// SIMATIC STEP 7 (V5.x) project MeM840D
// CPU: CPU 314
// station: P_ADR_BUS
// station: Hardware
// station: SIMATIC 300(1)
// program: Programma S7(1)

SYMBOL_TABLE
"POR_SX"	I 34.0	BOOL	// PORTA SX
"POR_DX"	I 34.1	BOOL	// PORTA DX
"CON_AVA"	I 40.4	BOOL	// CONTROPUNTA AVANTI
"CON_IND"	I 40.5	BOOL	// CONTROPUNTA INDIETRO
"BLKMOV"	SFC 20	SFC 20	// Copy Variables
"FILL"	SFC 21	SFC 21	// Initialize a Memory Area
"CREAT_DB"	SFC 22	SFC 22	// Create Data Block
"DIS_AIRT"	SFC 41	SFC 41	// Delay the Higher Priority Interrupts and Asynchronous Errors
"EN_AIRT"	SFC 42	SFC 42	// Enable Higher Priority Interrupts and Asynchronous Errors
"STP"	SFC 46	SFC 46	// Change the CPU to STOP
"WAIT"	SFC 47	SFC 47	// Delay Execution of the User Program
"RDSYSST"	SFC 51	SFC 51	// Read a System Status List or Partial List
"WR_USMSG"	SFC 52	SFC 52	// Write a User-Defined Diagnostic Event to the Diagnostic Buffer
"TIME_TCK"	SFC 64	SFC 64	// Read the System Time
END_SYMBOL_TABLE

// FB 1: know-how protected block, not included

// FB 2: know-how protected block, not included

// FB 3: know-how protected block, not included

// FB 4: know-how protected block, not included

// FB 5: know-how protected block, not included

// FB 6: know-how protected block, not included

// FB 7: know-how protected block, not included

FUNCTION_BLOCK FB 15
VERSION : 0.0
BEGIN
// body was compiled from another editor; compiled code not shown
END_FUNCTION_BLOCK

// FB 16: know-how protected block, not included

// FB 17: know-how protected block, not included

// FB 18: know-how protected block, not included

// FB 19: know-how protected block, not included

FUNCTION_BLOCK FB 20
VERSION : 2.2
BEGIN
// (block stored without names or comments; labels and parameter names are numbered)
NETWORK
TITLE =
      L     DW#16#87000000;
      LAR1;
      L     80;
      L     W#16#A000;
      +I;
      T     LW 0;
      A      [AR1,P#8.0];
      =     L 0.0;
      L     W [AR1,P#0.0];
      T     LW 2;
      L     W [AR1,P#6.0];
      SLD   16;
      L     B [AR1,P#4.0];
      OD;
      T     LD 4;
      CALL  "WR_USMSG" (
           SEND                     := FALSE,
           EVENTN                   := LW 0,
           INFO1                    := P#L 2.0 INT 1,
           INFO2                    := P#L 4.0 DINT 1,
           RET_VAL                  := LW 8);
END_FUNCTION_BLOCK

// FB 28: know-how protected block, not included

FUNCTION_BLOCK FB 120
AUTHOR : USER
VERSION : 0.2
BEGIN
// (block stored without names or comments; labels and parameter names are numbered)
NETWORK
TITLE =
      A     DIX [AR2,P#0.0];
      S     DIX [AR2,P#8.0];
      S     DIX [AR2,P#12.0];
NETWORK
TITLE =
      CALL  FB 3 , DB 91 (
           DIX 0.0                  := DBX [AR2,P#8.0],
           DIW 2                    := 1,
           DIW 4                    := W#16#1002,
           DIW 6                    := 10,
           DIW 8                    := 70,
           DID 10                   := P#DBX 0.0,
           DIX 132.0                := DBX [AR2,P#8.1],
           DIX 132.1                := DBX [AR2,P#8.2],
           DIX 134.0                := DBW [AR2,P#10.0],
           DIW 136                  := W#16#1001,
           DIW 138                  := 1,
           DIW 140                  := DBNO,
           DID 142                  := DBNO);
      A     DIX [AR2,P#8.1];
      =     DIX [AR2,P#2.0];
      R     DIX [AR2,P#8.0];
      A     DIX [AR2,P#8.2];
      =     DIX [AR2,P#2.1];
      R     DIX [AR2,P#8.0];
      L     DIW [AR2,P#10.0];
      T     DIW [AR2,P#4.0];
      A     DIX [AR2,P#8.2];
      AN    DB10.DBX 106.1;
      O     M 110.3;
      L     S5T#500MS;
      SP    T 121;
      A     T 121;
      =     M 110.3;
      A     M 110.3;
      FN    M 110.4;
      S     DIX [AR2,P#6.0];
      A     DB21.DBX 35.7;
      FP    M 110.6;
      A     M 110.6;
      R     DIX [AR2,P#6.0];
NETWORK
TITLE =
      AN    DIX [AR2,P#12.0];
      JC    M002;
      L     W#16#4C;
      +     1;
      T     DIW [AR2,P#14.0];
      OPN   DB 82;
      L     W#16#0;
      SLD   3;
      LAR1;
M001: L     W#16#0;
      T     DBB [AR1,P#0.0];
      +AR1  P#1.0;
      L     DIW [AR2,P#14.0];
      +     -1;
      T     DIW [AR2,P#14.0];
      LOOP  M001;
      SET;
      S     DB82.DBX 4.0;
      S     DB82.DBX 6.0;
      S     DB82.DBX 8.0;
      S     DB82.DBX 10.0;
      R     DIX [AR2,P#12.0];
M002: BE;
END_FUNCTION_BLOCK

// FC 1: know-how protected block, not included

// FC 2: know-how protected block, not included

// FC 3: know-how protected block, not included

// FC 4: know-how protected block, not included

// FC 6: know-how protected block, not included

// FC 7: know-how protected block, not included

// FC 8: know-how protected block, not included

// FC 9: know-how protected block, not included

// FC 10: know-how protected block, not included

// FC 11: know-how protected block, not included

FUNCTION FC 12 : VOID
AUTHOR : NUMERIK
FAMILY : _800D
NAME : Basics
VERSION : 4.0
BEGIN
// (block stored without names or comments; labels and parameter names are numbered)
END_FUNCTION

// FC 13: know-how protected block, not included

// FC 14: know-how protected block, not included

// FC 15: know-how protected block, not included

// FC 16: know-how protected block, not included

// FC 17: know-how protected block, not included

// FC 18: know-how protected block, not included

FUNCTION FC 19 : VOID
AUTHOR : NUMERIK
FAMILY : _800D
NAME : MCP_IFM
VERSION : 5.1
BEGIN
// (block stored without names or comments; labels and parameter names are numbered)
NETWORK
TITLE =
// (network holds code this reader does not know; not shown)
END_FUNCTION

// FC 20: know-how protected block, not included

// FC 21: know-how protected block, not included

// FC 22: know-how protected block, not included

FUNCTION FC 24 : VOID
AUTHOR : NUMERIK
FAMILY : _800D
NAME : MCP_IFM2
VERSION : 5.1
BEGIN
// (block stored without names or comments; labels and parameter names are numbered)
NETWORK
TITLE =
// (network holds code this reader does not know; not shown)
END_FUNCTION

FUNCTION FC 25 : VOID
AUTHOR : NUMERIK
FAMILY : _800D
NAME : MCP_IFT
VERSION : 5.1
BEGIN
// (block stored without names or comments; labels and parameter names are numbered)
NETWORK
TITLE =
// (network holds code this reader does not know; not shown)
END_FUNCTION

FUNCTION FC 26 : VOID
AUTHOR : NUMERIK
FAMILY : _800D
NAME : HPU_MCP
VERSION : 6.1
BEGIN
// (block stored without names or comments; labels and parameter names are numbered)
NETWORK
TITLE =
// (network holds code this reader does not know; not shown)
END_FUNCTION

FUNCTION FC 30 : VOID
VERSION : 0.0
BEGIN
// body was compiled from another editor; compiled code not shown
END_FUNCTION

FUNCTION FC 31 : VOID
VERSION : 0.0
BEGIN
// body was compiled from another editor; compiled code not shown
END_FUNCTION

FUNCTION FC 32 : VOID
VERSION : 0.0
BEGIN
// body was compiled from another editor; compiled code not shown
END_FUNCTION

FUNCTION FC 33 : VOID
VERSION : 0.0
BEGIN
// body was compiled from another editor; compiled code not shown
END_FUNCTION

// FC 34: know-how protected block, not included

// FC 35: know-how protected block, not included

FUNCTION FC 52 : VOID
AUTHOR : Zagorski
NAME : GENFUNK
VERSION : 0.15
BEGIN
// (block stored without names or comments; labels and parameter names are numbered)
NETWORK
TITLE =
      A     I 33.0;
      =     DB31.DBX 12.7;
      A     M 129.1;
      JC    M001;
      A     I 33.1;
      A     DB32.DBX 64.7;
      FN    M 15.0;
      =     M 15.1;
      A     I 33.1;
      S     M 15.2;
      A     M 15.1;
      R     M 15.2;
      A     M 15.2;
      =     DB32.DBX 12.7;
      JU    M002;
M001: A     I 6.7;
      A     I 2.7;
      AN    M 16.4;
      =     M 16.5;
      A     I 6.7;
      A     I 2.7;
      =     M 16.4;
      A     M 16.5;
      A     Q 4.7;
      R     M 16.6;
      A     M 16.5;
      AN    Q 4.7;
      S     M 16.6;
      A     M 16.6;
      =     Q 4.7;
      A     M 16.6;
      =     DB32.DBX 2.5;
      A     M 16.6;
      S     M 16.7;
      A     DB32.DBX 60.4;
      ON    M 16.6;
      R     M 16.7;
      L     PIW 32;
      T     MW 17;
      L     PIB 34;
      T     MB 19;
      A     M 18.1;
      A     DB32.DBX 64.7;
      FN    M 15.0;
      =     M 15.1;
      A     M 18.1;
      S     M 15.2;
      A     M 15.1;
      R     M 15.2;
      A     M 19.5;
      A     DB32.DBX 64.7;
      FN    M 15.4;
      =     M 15.5;
      A     M 19.5;
      S     M 15.6;
      A     M 15.5;
      R     M 15.6;
      A     M 16.6;
      A     M 15.6;
      O;
      AN    M 16.6;
      A     M 15.2;
      =     DB32.DBX 12.7;
M002: O     I 3.7;
      ON    I 32.0;
      =     M 75.1;
      O     I 3.7;
      ON    I 32.0;
      =     M 75.1;
      A     DB10.DBX 108.7;
      A(;
      O     I 32.0;
      O;
      A     I 3.7;
      A     I 4.4;
      A     Q 4.3;
      A     Q 0.4;
      );
      =     Q 36.4;
      A     DB10.DBX 108.7;
      =     Q 36.0;
      AN    I 32.0;
      A(;
      ON    I 3.7;
      ON    I 4.4;
      ON    Q 4.3;
      ON    Q 0.4;
      );
      =     DB10.DBX 56.1;
      A     I 32.0;
      O(;
      A     I 3.7;
      A     I 4.4;
      A     Q 4.3;
      A     Q 0.4;
      );
      AN    DB10.DBX 56.1;
      =     DB10.DBX 56.2;
NETWORK
TITLE =
      A     I 32.0;
      A     M 39.0;
      O;
      AN    DB33.DBX 61.4;
      A(;
      ON    M 39.0;
      ON    I 32.0;
      );
      O;
      A     I 3.7;
      A     I 4.4;
      A     Q 4.3;
      A     Q 0.4;
      =     DB31.DBX 2.1;
      =     DB31.DBX 21.7;
      =     DB32.DBX 2.1;
      =     DB32.DBX 21.7;
      =     DB33.DBX 2.1;
      =     DB33.DBX 21.7;
      A     M 51.0;
      =     DB21.DBX 25.3;
      =     DB31.DBX 1.5;
      =     DB32.DBX 1.5;
      =     DB33.DBX 1.6;
NETWORK
TITLE =
      A     I 5.5;
      A(;
      O     I 3.6;
      O     I 4.4;
      );
      =     M 40.4;
NETWORK
TITLE =
      A     M 40.4;
      A(;
      O     I 32.0;
      O;
      A     I 3.7;
      A     I 4.4;
      A     Q 4.3;
      A     Q 0.4;
      );
      S     M 39.0;
NETWORK
TITLE =
      O;
      A     I 4.2;
      A     DB33.DBX 61.4;
      AN    DB21.DBX 35.5;
      AN    DB21.DBX 35.0;
      O;
      AN    I 32.0;
      A(;
      ON    I 3.7;
      ON    I 4.4;
      ON    Q 4.3;
      ON    Q 0.4;
      );
      O     M 75.2;
      R     M 39.0;
NETWORK
TITLE =
      A     M 39.0;
      =     Q 3.6;
      AN    M 39.0;
      =     Q 2.5;
NETWORK
TITLE =
      A     M 39.0;
      A     I 32.0;
      O;
      A     I 3.7;
      A     I 4.4;
      A     Q 4.3;
      A     Q 0.4;
      S     Q 37.7;
      A     DB33.DBX 61.4;
      A(;
      ON    M 39.0;
      ON    I 32.0;
      );
      A(;
      ON    I 3.7;
      ON    I 4.4;
      ON    Q 4.3;
      ON    Q 0.4;
      );
      R     Q 37.7;
NETWORK
TITLE =
      A     I 32.0;
      FN    M 3.1;
      =     M 3.2;
      A     M 3.2;
      S     M 3.0;
      A     I 3.7;
      R     M 3.0;
NETWORK
TITLE =
      L     DB82.DBB 45;
      L     0;
      ==I;
      =     M 38.0;
NETWORK
TITLE =
      L     DB82.DBB 45;
      L     3;
      <=I;
      =     M 38.6;
NETWORK
TITLE =
      A     DB33.DBX 82.3;
      =     DB82.DBX 16.6;
      A     DB33.DBX 82.3;
      A     DB33.DBX 61.4;
      S     M 40.0;
      A     DB33.DBX 16.3;
      R     M 40.0;
      A     M 40.0;
      =     DB33.DBX 18.5;
      AN    M 40.0;
      JC    M003;
      A     DB33.DBX 82.0;
      AN    DB33.DBX 82.1;
      AN    DB33.DBX 82.2;
      S     Q 36.1;
      R     Q 36.2;
      AN    DB33.DBX 82.0;
      A     DB33.DBX 82.1;
      AN    DB33.DBX 82.2;
      S     Q 36.2;
      R     Q 36.1;
M003: A     I 33.6;
      AN    I 33.7;
      S     DB33.DBX 16.0;
      R     DB33.DBX 16.1;
      R     DB33.DBX 16.2;
      AN    I 33.6;
      A     I 33.7;
      R     DB33.DBX 16.0;
      S     DB33.DBX 16.1;
      R     DB33.DBX 16.2;
      A     DB33.DBX 16.0;
      =     M 41.0;
      A     DB33.DBX 16.1;
      =     M 41.1;
      A     DB33.DBX 16.2;
      =     M 41.2;
      A     DB33.DBX 82.0;
      =     M 42.0;
      A     DB33.DBX 82.1;
      =     M 42.1;
      A     DB33.DBX 82.2;
      =     M 42.2;
      L     MB 41;
      L     MB 42;
      ==I;
      =     M 40.1;
      A     M 40.1;
      L     S5T#2S;
      SD    T 70;
      A     T 70;
      =     M 40.2;
      A     M 40.2;
      A     M 40.0;
      S     M 40.3;
      AN    M 40.0;
      R     M 40.3;
      A     M 40.3;
      =     DB33.DBX 16.3;
      AN    M 40.0;
      L     S5T#4S;
      SP    T 69;
NETWORK
TITLE =
      O     I 7.1;
      AN    DB21.DBX 35.0;
      AN    DB21.DBX 35.1;
      =     DB33.DBX 4.7;
      =     Q 5.1;
      AN    I 7.1;
      L     S5T#4S;
      SP    T 68;
NETWORK
TITLE =
      A     I 3.7;
      A     I 4.4;
      A     Q 4.3;
      A     Q 0.4;
      A(;
      A     DB82.DBX 40.0;
      A     M 38.0;
      O;
      AN    DB82.DBX 40.0;
      A     DB11.DBX 6.2;
      );
      =     Q 37.3;
NETWORK
TITLE =
      A     DB33.DBX 61.4;
      L     S5T#4S;
      SF    T 55;
      NOP   0;
      NOP   0;
      NOP   0;
      NOP   0;
NETWORK
TITLE =
      A(;
      O     Q 5.1;
      O     T 68;
      O     M 40.0;
      O     T 69;
      );
      A(;
      A     DB82.DBX 40.0;
      AN    DB82.DBX 41.5;
      O;
      AN    DB82.DBX 40.0;
      AN    DB21.DBX 35.0;
      );
      O;
      A(;
      A(;
      A     DB82.DBX 40.0;
      A     M 38.0;
      O;
      AN    DB82.DBX 40.0;
      A(;
      O     DB11.DBX 6.2;
      O     DB11.DBX 7.2;
      O     DB11.DBX 6.1;
      );
      O;
      A     T 55;
      A(;
      A     DB82.DBX 40.0;
      AN    DB82.DBX 41.5;
      O;
      AN    DB82.DBX 40.0;
      AN    DB21.DBX 35.0;
      O     DB21.DBX 33.7;
      O     DB21.DBX 33.4;
      O;
      A     DB82.DBX 40.0;
      A     DB82.DBX 41.6;
      A     Q 1.4;
      A     Q 1.6;
      A(;
      O     Q 2.0;
      O     Q 3.4;
      );
      O;
      A     DB82.DBX 40.0;
      A     DB82.DBX 41.6;
      A     DB21.DBX 32.5;
      A     Q 1.4;
      O;
      AN    DB82.DBX 40.0;
      A     DB21.DBX 35.2;
      A     Q 1.4;
      A     Q 1.6;
      A     Q 2.0;
      );
      );
      AN    M 3.0;
      O;
      A     I 3.7;
      A     M 3.0;
      );
      A(;
      O     Q 2.0;
      O     Q 3.4;
      O;
      A     DB33.DBX 61.4;
      A     DB21.DBX 32.5;
      );
      =     Q 37.4;
NETWORK
TITLE =
NETWORK
TITLE =
      A(;
      A     DB82.DBX 40.0;
      A     M 38.0;
      O;
      AN    DB82.DBX 40.0;
      A     DB11.DBX 6.2;
      );
      A     I 4.4;
      =     M 16.1;
NETWORK
TITLE =
      AN    "POR_SX";
      AN    "POR_DX";
      AN    I 34.2;
      A(;
      AN    M 45.0;
      AN    M 45.1;
      O     M 134.0;
      O     M 134.1;
      );
      JC    M004;
      A     M 51.0;
      AN    Q 5.1;
      AN    M 40.0;
      S     DB33.DBX 4.3;
      S     DB82.DBX 10.1;
      R     DB82.DBX 10.0;
      AN    Q 5.1;
      AN    M 40.0;
      AN    DB21.DBX 32.5;
      R     I 2.4;
      A     DB33.DBX 61.4;
      AN    Q 5.1;
      AN    M 40.0;
      S     M 71.0;
      A     M 71.0;
      AN    Q 5.1;
      AN    T 68;
      AN    M 40.0;
      AN    T 69;
      R     DB33.DBX 21.7;
M004: AN    "POR_SX";
      AN    "POR_DX";
      AN    I 34.2;
      A(;
      AN    M 45.0;
      AN    M 45.1;
      O     M 134.0;
      O     M 134.1;
      );
      R     M 71.0;
NETWORK
TITLE =
      AN    "POR_SX";
      AN    "POR_DX";
      A(;
      ON    DB33.DBX 61.4;
      O;
      A(;
      A     DB82.DBX 40.0;
      AN    M 38.0;
      O;
      AN    DB82.DBX 40.0;
      AN    DB11.DBX 6.2;
      AN    DB11.DBX 7.2;
      AN    DB11.DBX 6.1;
      );
      A(;
      O     DB21.DBX 35.5;
      O     DB21.DBX 35.0;
      );
      O;
      A     DB82.DBX 40.0;
      AN    M 38.0;
      A     DB82.DBX 41.6;
      AN    DB21.DBX 32.5;
      A(;
      ON    Q 1.4;
      ON    Q 1.6;
      O;
      AN    Q 2.0;
      AN    Q 3.4;
      );
      O;
      AN    DB82.DBX 40.0;
      AN    DB11.DBX 6.2;
      AN    DB11.DBX 7.2;
      AN    DB11.DBX 6.1;
      A     DB21.DBX 35.2;
      AN    DB21.DBX 32.5;
      A(;
      ON    Q 1.4;
      ON    Q 1.6;
      ON    Q 2.0;
      );
      );
      =     Q 36.3;
NETWORK
TITLE =
      AN    DB82.DBX 40.0;
      A     I 3.7;
      =     DB33.DBX 2.2;
NETWORK
TITLE =
      O     "POR_SX";
      O     "POR_DX";
      A(;
      A     DB82.DBX 40.0;
      AN    M 38.6;
      O;
      AN    DB82.DBX 40.0;
      AN    DB11.DBX 6.2;
      AN    DB11.DBX 7.2;
      AN    DB11.DBX 6.1;
      );
      O     I 34.2;
      =     M 38.7;
      O     M 38.7;
      O;
      AN    I 41.7;
      AN    M 16.1;
      =     DB21.DBX 7.0;
      S     DB21.DBX 6.1;
      S     DB21.DBX 6.0;
      S     DB21.DBX 7.3;
NETWORK
TITLE =
      A     M 126.0;
      JC    M005;
      A     M 76.2;
      AN    M 75.3;
      A(;
      A     DB82.DBX 40.0;
      AN    M 38.0;
      O;
      AN    DB82.DBX 40.0;
      AN    DB11.DBX 6.2;
      AN    DB11.DBX 7.2;
      );
      S     DB21.DBX 6.1;
M005: NOP   0;
NETWORK
TITLE =
      A     M 126.0;
      JC    M006;
      A     M 51.0;
      A     M 76.2;
      AN    M 75.3;
      A(;
      A     DB82.DBX 40.0;
      AN    M 38.0;
      O;
      AN    DB82.DBX 40.0;
      AN    DB11.DBX 6.2;
      AN    DB11.DBX 7.2;
      );
      S     DB21.DBX 6.0;
M006: NOP   0;
NETWORK
TITLE =
      A     I 34.2;
      =     DB2.DBX 180.0;
      A     I 35.4;
      =     DB2.DBX 180.3;
      A     M 12.7;
      =     DB2.DBX 180.5;
      A     T 66;
      =     DB2.DBX 180.6;
      A(;
      O     M 134.2;
      O     M 134.3;
      O     M 134.4;
      );
      A(;
      O     M 45.0;
      O     M 45.1;
      AN    DB33.DBX 4.7;
      AN    M 40.0;
      AN    I 4.4;
      );
      A(;
      ON    DB33.DBX 61.4;
      O     I 2.5;
      O     I 5.4;
      O     I 4.0;
      O     I 2.1;
      );
      =     DB2.DBX 180.7;
      A     M 134.0;
      AN    I 35.0;
      =     DB2.DBX 181.0;
      AN    I 35.1;
      =     DB2.DBX 181.1;
      AN    I 35.2;
      =     DB2.DBX 181.2;
      AN    M 134.0;
      AN    I 35.0;
      =     DB2.DBX 181.3;
      AN    I 35.6;
      =     DB2.DBX 181.4;
      AN    I 35.7;
      =     DB2.DBX 181.5;
      AN    M 125.0;
      AN    I 35.5;
      =     DB2.DBX 181.6;
      AN    M 39.0;
      =     DB2.DBX 185.0;
      AN    M 40.0;
      A(;
      AN    I 33.6;
      AN    I 33.7;
      O;
      A     I 33.6;
      A     I 33.7;
      );
      =     DB2.DBX 185.2;
      JU    M007;
      A(;
      O     "POR_SX";
      O     "POR_DX";
      );
      A(;
      A     DB82.DBX 40.0;
      AN    M 38.6;
      O;
      AN    DB82.DBX 40.0;
      AN    DB11.DBX 6.2;
      AN    DB11.DBX 7.2;
      AN    DB11.DBX 6.1;
      );
      A(;
      O     I 2.5;
      O     I 5.4;
      O     I 4.0;
      O     I 2.1;
      );
      S     M 15.3;
      A(;
      AN    "POR_SX";
      AN    "POR_DX";
      O;
      A     DB82.DBX 40.0;
      A     M 38.6;
      O;
      AN    DB82.DBX 40.0;
      A(;
      O     DB11.DBX 6.2;
      O     DB11.DBX 7.2;
      O     DB11.DBX 6.1;
      );
      );
      O     M 75.1;
      O     I 2.4;
      O     I 5.3;
      R     M 15.3;
      A     "POR_SX";
      A(;
      O     M 10.3;
      ON    M 38.7;
      );
      A     M 15.3;
      A(;
      A     DB82.DBX 40.0;
      AN    M 38.6;
      O;
      AN    DB82.DBX 40.0;
      AN    DB11.DBX 6.2;
      AN    DB11.DBX 7.2;
      AN    DB11.DBX 6.1;
      );
      =     DB2.DBX 185.3;
      A     "POR_DX";
      A(;
      O     M 10.3;
      ON    M 38.7;
      );
      A     M 15.3;
      A(;
      A     DB82.DBX 40.0;
      AN    M 38.6;
      O;
      AN    DB82.DBX 40.0;
      AN    DB11.DBX 6.2;
      AN    DB11.DBX 7.2;
      AN    DB11.DBX 6.1;
      );
      =     DB2.DBX 185.4;
      A     M 38.7;
      AN    M 10.3;
      A     M 15.3;
      =     DB2.DBX 185.5;
M007: NOP   0;
      A(;
      O     "POR_SX";
      O     "POR_DX";
      );
      A(;
      O     I 2.5;
      O     I 5.4;
      O     I 4.0;
      O     I 2.1;
      );
      S     M 15.3;
      AN    "POR_SX";
      AN    "POR_DX";
      O     M 75.1;
      O     I 2.4;
      O     I 5.3;
      R     M 15.3;
      A     "POR_SX";
      A(;
      O     M 10.3;
      ON    M 38.7;
      );
      A     M 15.3;
      =     DB2.DBX 185.3;
      A     "POR_DX";
      A(;
      O     M 10.3;
      ON    M 38.7;
      );
      A     M 15.3;
      =     DB2.DBX 185.4;
      A     M 38.7;
      AN    M 10.3;
      A     M 15.3;
      =     DB2.DBX 185.5;
      A     M 126.0;
      JC    M008;
      A     M 76.3;
      =     DB2.DBX 180.1;
      A     M 76.7;
      =     DB2.DBX 180.2;
      A(;
      O     Q 37.0;
      O     Q 37.1;
      );
      A     I 33.3;
      L     S5T#80MS;
      SD    T 87;
      NOP   0;
      NOP   0;
      NOP   0;
      NOP   0;
      A     I 32.0;
      A     T 87;
      S     M 76.6;
      A     M 75.1;
      R     M 76.6;
      A     M 76.6;
      =     DB2.DBX 185.7;
      A     M 75.4;
      AN    M 77.4;
      =     DB2.DBX 186.0;
      A     M 77.5;
      =     DB2.DBX 186.1;
      AN    M 88.4;
      AN    M 77.5;
      AN    T 87;
      =     DB2.DBX 186.2;
      AN    M 77.4;
      AN    M 75.4;
      AN    M 77.5;
      AN    T 87;
      =     DB2.DBX 186.3;
M008: NOP   0;
      A     M 129.1;
      A     M 16.7;
      =     DB2.DBX 186.4;
      A(;
      O     M 134.2;
      O     M 134.4;
      );
      A(;
      A     Q 38.6;
      A     M 46.7;
      O;
      A     Q 38.5;
      AN    M 46.7;
      );
      =     DB2.DBX 186.5;
      A(;
      O     M 134.3;
      O     M 134.4;
      );
      A     Q 38.3;
      AN    M 44.0;
      =     DB2.DBX 186.6;
      A(;
      O     M 134.2;
      O     M 134.4;
      );
      AN    M 45.4;
      A(;
      O     I 40.0;
      O     I 40.1;
      );
      O;
      A(;
      O     M 134.3;
      O     M 134.4;
      );
      AN    M 45.5;
      A(;
      O     "CON_AVA";
      O     "CON_IND";
      );
      =     DB2.DBX 186.7;
      A(;
      O     M 134.2;
      O     M 134.4;
      );
      A(;
      A     Q 38.5;
      AN    Q 38.6;
      AN    I 34.6;
      );
      A     Q 36.4;
      =     DB2.DBX 187.0;
      A(;
      O     M 134.3;
      O     M 134.4;
      );
      AN    I 41.0;
      A     Q 38.0;
      A     Q 36.4;
      =     DB2.DBX 187.1;
      A(;
      O     M 134.2;
      O     M 134.4;
      );
      A     M 45.1;
      =     DB2.DBX 187.2;
      JU    M009;
      A     M 72.1;
      A     M 72.0;
      L     S5T#4S;
      SD    T 73;
      A     T 73;
      =     DB2.DBX 187.3;
      AN    M 72.1;
      A     M 72.0;
      L     S5T#4S;
      SD    T 74;
      A     T 74;
      =     DB2.DBX 187.4;
M009: NOP   0;
      AN    I 32.1;
      A     M 39.0;
      =     DB2.DBX 192.0;
      AN    I 41.7;
      =     DB2.DBX 194.0;
      A(;
      ON    M 43.7;
      O     M 43.5;
      ON    DB11.DBX 6.2;
      O     DB21.DBX 35.0;
      O     DB21.DBX 35.1;
      );
      A     I 4.4;
      A     I 6.7;
      =     DB2.DBX 194.4;
NETWORK
TITLE =
      A     M 75.2;
      R     M 10.0;
      R     M 10.2;
      R     M 10.6;
      O(;
      A     DB31.DBX 76.0;
      FN    M 11.0;
      );
      O(;
      A     DB31.DBX 76.0;
      FP    M 11.1;
      );
      =     M 11.2;
      O(;
      A     DB32.DBX 76.0;
      FN    M 10.4;
      );
      O(;
      A     DB32.DBX 76.0;
      FP    M 10.5;
      );
      =     M 10.7;
      AN    M 10.6;
      L     S5T#2S;
      SD    T 64;
      A     T 64;
      =     M 10.6;
      A     M 10.0;
      O     M 11.2;
      O     M 10.7;
      L     C#600;
      S     C 1;
      A     M 10.6;
      A     DB31.DBX 61.4;
      A     DB32.DBX 61.4;
      CD    C 1;
      L     C 1;
      L     0;
      ==I;
      =     M 10.0;
      A     M 10.0;
      O     M 11.2;
      O     M 10.7;
      L     S5T#10S;
      SE    T 61;
      A     T 61;
      =     M 10.1;
      AN    M 10.2;
      L     S5T#4S;
      SE    T 62;
      A     T 62;
      =     M 10.2;
      A     M 10.2;
      L     S5T#2S;
      SE    T 63;
      A     T 63;
      =     M 10.3;
      A     M 10.1;
      A     M 10.6;
      AN    M 14.5;
      S     M 14.2;
      O     M 14.4;
      O     T 59;
      O;
      A     M 12.7;
      A(;
      O     M 75.1;
      O     M 75.2;
      );
      R     M 14.2;
      A     M 14.2;
      A     I 35.3;
      L     S5T#1S;
      SE    T 60;
      A     T 60;
      FN    M 14.3;
      =     M 14.4;
      A     M 14.4;
      S     M 14.5;
      A     T 59;
      R     M 14.5;
      A     M 14.5;
      AN    I 35.3;
      L     S5T#1S;
      SE    T 59;
      A     I 7.7;
      AN    I 35.3;
      S     M 14.0;
      A     M 14.0;
      A     I 7.7;
      A     I 35.3;
      S     M 14.1;
      A     M 14.0;
      A     M 14.1;
      L     S5T#2S;
      SE    T 67;
      O     T 67;
      ON    I 7.7;
      R     M 14.0;
      R     M 14.1;
      A(;
      A     M 14.2;
      A(;
      O     M 10.1;
      ON    M 14.2;
      ON    M 12.7;
      );
      O;
      AN    I 35.3;
      A     I 7.7;
      AN    T 67;
      );
      A     I 32.0;
      =     Q 36.6;
      =     Q 5.7;
      A     M 10.1;
      A     I 35.3;
      FN    M 11.4;
      =     M 11.5;
      A     M 10.1;
      A     I 35.3;
      FP    M 11.6;
      =     M 11.7;
      A     M 10.1;
      A     Q 36.6;
      FN    M 12.0;
      =     M 12.1;
      A     M 10.1;
      A     Q 36.6;
      FP    M 12.2;
      =     M 12.3;
      AN    I 7.7;
      A(;
      O     M 12.1;
      O     M 12.3;
      );
      AN    M 12.4;
      S     M 12.5;
      AN    I 7.7;
      A(;
      O     M 11.5;
      O     M 11.7;
      );
      A     M 12.4;
      S     M 12.6;
      O     M 12.1;
      O     M 12.3;
      S     M 12.4;
      AN    M 10.1;
      AN    Q 36.6;
      R     M 12.4;
      A     M 12.5;
      A     M 12.6;
      AN    M 10.1;
      A     M 10.3;
      O     M 75.1;
      O     M 75.2;
      R     M 12.4;
      R     M 12.5;
      R     M 12.6;
      R     M 12.7;
      A     M 12.5;
      AN    M 12.6;
      AN    M 10.1;
      S     M 12.7;
NETWORK
TITLE =
      A     Q 36.4;
      A     I 35.0;
      L     S5T#5S;
      SD    T 65;
      AN    I 34.3;
      A     T 65;
      L     S5T#5S;
      SD    T 66;
NETWORK
TITLE =
      A     I 7.5;
      AN    M 70.0;
      =     M 70.1;
      A     I 7.5;
      =     M 70.0;
      A     M 70.1;
      O     DB21.DBX 195.1;
      O     DB21.DBX 197.6;
      A     Q 36.5;
      ON    I 32.0;
      R     M 70.2;
      A     M 70.1;
      O     DB21.DBX 194.7;
      A     I 32.0;
      AN    Q 36.5;
      S     M 70.2;
      A     M 70.2;
      A     I 35.1;
      =     Q 36.5;
      =     Q 5.5;
NETWORK
TITLE =
      A     M 125.0;
      JC    M010;
      CALL  FC 70;
M010: NOP   0;
NETWORK
TITLE =
      A     I 5.0;
      AN    M 70.4;
      =     M 70.5;
      A     I 5.0;
      =     M 70.4;
      A     M 70.5;
      A     Q 37.6;
      R     M 70.6;
      A     M 70.5;
      AN    Q 37.6;
      S     M 70.6;
      A     M 70.6;
      =     Q 37.6;
      =     Q 3.1;
NETWORK
TITLE =
      A     DB82.DBX 40.0;
      AN    DB33.DBX 94.6;
      A     DB21.DBX 316.0;
      FN    M 111.0;
      S     DB2.DBX 145.0;
      A     DB33.DBX 83.5;
      R     DB2.DBX 145.0;
      A     DB2.DBX 145.0;
      S     DB21.DBX 6.0;
NETWORK
TITLE =
NETWORK
TITLE =
      AN    DB82.DBX 40.0;
      S     DB10.DBX 57.0;
END_FUNCTION

FUNCTION FC 60 : VOID
AUTHOR : ZAGORSKI
NAME : HYDRCS
VERSION : 0.2
BEGIN
// (block stored without names or comments; labels and parameter names are numbered)
NETWORK
TITLE =
      A     M 134.0;
      JC    M001;
NETWORK
TITLE =
      A     I 34.4;
      A     M 39.0;
      =     M 39.4;
NETWORK
TITLE =
      A     I 5.5;
      A(;
      O     I 3.6;
      O     I 4.4;
      );
      =     M 40.4;
NETWORK
TITLE =
      A     M 40.4;
      A     M 51.0;
      A(;
      O     I 32.0;
      O;
      A     I 3.7;
      A     I 4.4;
      A     Q 4.3;
      A     Q 0.4;
      );
      S     M 39.0;
NETWORK
TITLE =
      AN    M 39.4;
      L     S5T#1S;
      SD    T 35;
      NOP   0;
      NOP   0;
      NOP   0;
      NOP   0;
NETWORK
TITLE =
      A     M 39.0;
      L     S5T#5S;
      SP    T 30;
      NOP   0;
      NOP   0;
      NOP   0;
      NOP   0;
NETWORK
TITLE =
      A(;
      A     I 4.2;
      A     DB33.DBX 61.4;
      AN    DB21.DBX 35.5;
      AN    DB21.DBX 35.0;
      O;
      AN    I 32.0;
      A(;
      ON    I 3.7;
      ON    I 4.4;
      ON    Q 4.3;
      ON    Q 0.4;
      );
      O     M 75.2;
      ON    I 35.0;
      O;
      AN    T 30;
      A     T 35;
      );
      R     M 39.0;
      NOP   0;
      NOP   0;
NETWORK
TITLE =
      A     M 39.0;
      =     Q 36.4;
      =     Q 3.6;
      AN    M 39.0;
      =     Q 2.5;
NETWORK
TITLE =
M001: NOP   0;
NETWORK
TITLE =
      A     DB33.DBX 61.4;
      A(;
      O     DB11.DBX 6.2;
      O;
      AN    DB21.DBX 35.0;
      AN    DB21.DBX 35.5;
      A(;
      O     DB11.DBX 6.1;
      O     DB11.DBX 6.0;
      );
      );
      A     M 39.0;
      L     S5T#2S;
      SD    T 31;
      NOP   0;
      NOP   0;
      NOP   0;
      A     T 31;
      =     M 45.7;
NETWORK
TITLE =
      A     M 45.7;
      AN    I 40.0;
      AN    I 40.1;
      S     M 45.4;
      A(;
      ON    M 45.7;
      );
      R     M 45.4;
      NOP   0;
NETWORK
TITLE =
      A     M 45.7;
      AN    "CON_AVA";
      AN    "CON_IND";
      A(;
      O     "POR_SX";
      O     "POR_DX";
      );
      S     M 45.5;
      A(;
      ON    M 45.7;
      O;
      AN    "POR_SX";
      AN    "POR_DX";
      );
      R     M 45.5;
      NOP   0;
NETWORK
TITLE =
      A     I 6.7;
      AN    M 43.1;
      =     M 43.0;
NETWORK
TITLE =
      A     I 6.7;
      =     M 43.1;
NETWORK
TITLE =
      AN    Q 38.5;
      A     Q 38.6;
      A     I 34.4;
      AN    I 34.6;
      AN    I 40.3;
      A     I 40.2;
      A     M 46.7;
      O;
      A     Q 38.5;
      AN    Q 38.6;
      AN    I 34.4;
      A     I 34.6;
      A     I 40.3;
      AN    I 40.2;
      AN    M 46.7;
      =     M 43.7;
NETWORK
TITLE =
      A     Q 38.5;
      AN    Q 38.6;
      AN    I 34.4;
      A     I 34.6;
      A     I 40.3;
      AN    I 40.2;
      A     M 46.7;
      O;
      AN    Q 38.5;
      A     Q 38.6;
      A     I 34.4;
      AN    I 34.6;
      AN    I 40.3;
      A     I 40.2;
      AN    M 46.7;
      =     M 43.5;
NETWORK
TITLE =
      A     DB11.DBX 6.2;
      AN    DB21.DBX 35.0;
      AN    DB21.DBX 35.1;
      A     I 4.4;
      A     M 43.7;
      AN    M 43.5;
      A     M 43.0;
      A     M 46.7;
      R     M 46.6;
      A     DB11.DBX 6.2;
      AN    DB21.DBX 35.0;
      AN    DB21.DBX 35.1;
      A     I 4.4;
      A     M 43.7;
      AN    M 43.5;
      A     M 43.0;
      AN    M 46.7;
      S     M 46.6;
      A     M 46.6;
      =     M 46.7;
      A     M 51.0;
      =     M 46.7;
NETWORK
TITLE =
NETWORK
TITLE =
      A(;
      A     I 40.0;
      A     M 45.4;
      O     M 75.2;
      );
      S     M 43.2;
      A     I 40.1;
      A     M 45.4;
      R     M 43.2;
      NOP   0;
NETWORK
TITLE =
      AN    M 134.2;
      AN    M 134.4;
      O     M 134.0;
      O     M 134.1;
      JC    M002;
      A     M 43.2;
      A     M 46.7;
      O;
      AN    M 43.2;
      AN    M 46.7;
      =     Q 38.5;
      A     M 43.2;
      AN    M 46.7;
      O;
      AN    M 43.2;
      A     M 46.7;
      =     Q 38.6;
M002: NOP   0;
NETWORK
TITLE =
      A(;
      A(;
      O     M 134.2;
      O     M 134.4;
      );
      A(;
      A     Q 38.5;
      AN    Q 38.6;
      A     M 46.7;
      O;
      AN    Q 38.5;
      A     Q 38.6;
      AN    M 46.7;
      );
      A     M 43.2;
      L     S5T#6S;
      SD    T 32;
      NOP   0;
      NOP   0;
      NOP   0;
      A     T 32;
      );
      A     I 34.6;
      AN    I 40.2;
      AN    I 40.3;
      =     M 43.4;
NETWORK
TITLE =
NETWORK
TITLE =
      A(;
      A     "CON_AVA";
      A     M 45.5;
      O     M 75.2;
      );
      S     M 43.3;
      A     "CON_IND";
      A     M 45.5;
      R     M 43.3;
      NOP   0;
NETWORK
TITLE =
      AN    M 134.3;
      AN    M 134.4;
      O     M 134.0;
      O     M 134.1;
      JC    M003;
      A     M 43.3;
      =     Q 38.0;
      AN    M 43.3;
      =     Q 38.1;
M003: NOP   0;
NETWORK
TITLE =
      A(;
      O     M 134.3;
      O     M 134.4;
      );
      A(;
      A     Q 38.0;
      A     M 43.3;
      O;
      A     Q 38.1;
      AN    M 43.3;
      L     S5T#4S;
      SD    T 33;
      NOP   0;
      NOP   0;
      NOP   0;
      A     T 33;
      );
      A(;
      A     I 41.0;
      A     Q 38.0;
      AN    I 40.6;
      AN    I 40.7;
      O;
      A     Q 38.1;
      A     I 40.7;
      AN    I 40.6;
      );
      =     M 44.0;
NETWORK
TITLE =
NETWORK
TITLE =
      A(;
      O     M 43.4;
      O     M 134.0;
      O     M 134.1;
      O     M 134.3;
      );
      A(;
      O     M 44.0;
      O     M 134.0;
      O     M 134.1;
      O     M 134.2;
      );
      A     Q 36.4;
      =     M 44.4;
NETWORK
TITLE =
NETWORK
TITLE =
NETWORK
TITLE =
NETWORK
TITLE =
      A(;
      ON    I 34.4;
      O;
      A     Q 38.5;
      AN    Q 38.6;
      AN    I 34.6;
      );
      A(;
      O     M 134.2;
      O     M 134.4;
      );
      O;
      AN    I 41.0;
      A     Q 38.0;
      A(;
      O     M 134.3;
      O     M 134.4;
      );
      =     M 45.0;
NETWORK
TITLE =
      A(;
      O     I 40.2;
      O     I 40.3;
      );
      A(;
      O     M 134.2;
      O     M 134.4;
      );
      O;
      A(;
      O     M 134.3;
      O     M 134.4;
      );
      A     Q 38.0;
      A(;
      O     I 40.6;
      O     I 40.7;
      );
      =     M 45.1;
NETWORK
TITLE =
      A(;
      O     M 134.2;
      O     M 134.3;
      O     M 134.4;
      );
      A(;
      ON    M 44.4;
      O     M 45.0;
      );
      A(;
      A     DB82.DBX 40.0;
      AN    M 38.0;
      O;
      AN    DB82.DBX 40.0;
      AN    DB11.DBX 6.2;
      AN    DB11.DBX 7.2;
      );
      =     M 46.2;
      A     M 46.2;
      AN    DB82.DBX 37.3;
      AN    "POR_SX";
      AN    "POR_DX";
      S     M 46.0;
      A     M 75.1;
      R     M 46.0;
      NOP   0;
NETWORK
TITLE =
      A     M 46.0;
      S     DB21.DBX 6.1;
      NOP   0;
      NOP   0;
NETWORK
TITLE =
      A(;
      O     M 134.2;
      O     M 134.3;
      O     M 134.4;
      );
      A(;
      ON    M 44.4;
      O     M 45.0;
      );
      A(;
      A     DB82.DBX 40.0;
      AN    M 38.0;
      O;
      AN    DB82.DBX 40.0;
      AN    DB11.DBX 6.2;
      AN    DB11.DBX 7.2;
      );
      =     M 46.3;
      A     M 46.3;
      AN    DB82.DBX 37.3;
      AN    "POR_SX";
      AN    "POR_DX";
      S     M 46.1;
      A     M 75.1;
      R     M 46.1;
      NOP   0;
NETWORK
TITLE =
      A     M 46.1;
      S     DB21.DBX 6.0;
      NOP   0;
      NOP   0;
END_FUNCTION

FUNCTION FC 70 : VOID
VERSION : 0.1
BEGIN
// (block stored without names or comments; labels and parameter names are numbered)
NETWORK
TITLE =
      A     I 6.7;
      AN    M 71.1;
      =     M 71.2;
      A     I 6.7;
      =     M 71.1;
      A     M 71.2;
      O     DB21.DBX 197.6;
      A     Q 36.7;
      ON    I 32.0;
      R     M 71.3;
      A     M 71.2;
      AN    Q 36.7;
      A     I 32.0;
      S     M 71.3;
      A     M 71.3;
      A     I 35.5;
      =     Q 36.7;
      =     Q 4.7;
END_FUNCTION

FUNCTION FC 90 : VOID
AUTHOR : Tested
NAME : Logic
VERSION : 0.2
BEGIN
// (block stored without names or comments; labels and parameter names are numbered)
NETWORK
TITLE =
      O     DB21.DBX 35.0;
      O     DB82.DBX 41.5;
      O     DB82.DBX 41.6;
      A     Q 1.6;
      AN    Q 1.7;
      O;
      AN    DB21.DBX 35.0;
      AN    DB82.DBX 41.5;
      AN    DB82.DBX 41.6;
      O     M 38.0;
      =     M 90.5;
      O     DB21.DBX 35.0;
      O     DB82.DBX 41.5;
      O     DB82.DBX 41.6;
      AN    DB82.DBX 42.0;
      AN    Q 2.0;
      AN    Q 3.4;
      O;
      AN    DB21.DBX 35.0;
      AN    DB82.DBX 41.5;
      AN    DB82.DBX 41.6;
      O     M 38.0;
      =     M 90.6;
NETWORK
TITLE =
      A     DB82.DBX 41.3;
      A     DB82.DBX 41.6;
      A     Q 1.6;
      A(;
      O     Q 2.0;
      O     Q 3.4;
      );
      S     M 91.3;
      A     Q 2.1;
      A(;
      AN    "POR_SX";
      AN    "POR_DX";
      AN    I 34.2;
      AN    I 34.7;
      );
      O     M 75.1;
      R     M 91.3;
NETWORK
TITLE =
      A     DB82.DBX 41.4;
      A     DB82.DBX 41.6;
      A     Q 1.6;
      A(;
      O     Q 2.0;
      O     Q 3.4;
      );
      S     M 91.4;
      A     Q 2.1;
      A(;
      AN    "POR_SX";
      AN    "POR_DX";
      AN    I 34.2;
      AN    I 34.7;
      );
      O     M 75.1;
      R     M 91.4;
NETWORK
TITLE =
      L     IB 3;
      AW    W#16#1F;
      T     DB82.DBB 1;
      L     IB 0;
      SRW   4;
      T     DB82.DBB 2;
      A     I 2.1;
      AN    DB21.DBX 7.0;
      =     DB82.DBX 4.1;
      AN    I 2.1;
      =     DB82.DBX 4.0;
      AN    I 2.0;
      =     DB82.DBX 6.1;
      A     I 2.0;
      =     DB82.DBX 6.0;
      A     M 82.7;
      A     M 40.1;
      =     DB82.DBX 8.1;
      AN    M 82.7;
      ON    M 40.1;
      =     DB82.DBX 8.0;
      O     I 5.3;
      O     I 3.7;
      =     DB82.DBX 10.1;
      AN    I 5.3;
      AN    I 3.7;
      =     DB82.DBX 10.0;
      A     I 5.4;
      AN    M 91.3;
      AN    M 91.4;
      O;
      A     M 91.3;
      A     I 2.5;
      =     DB82.DBX 12.1;
      =     M 82.5;
      A     I 4.0;
      AN    M 91.3;
      AN    M 91.4;
      O;
      A     M 91.4;
      A     I 2.5;
      =     M 82.6;
      =     DB82.DBX 12.0;
      O     M 82.5;
      O     M 82.6;
      =     M 82.7;
      A     I 7.3;
      =     DB82.DBX 12.2;
      A     I 7.0;
      =     DB82.DBX 12.3;
      A     I 7.6;
      =     DB82.DBX 12.4;
      A     I 7.2;
      =     DB82.DBX 12.7;
      A     I 7.4;
      =     DB82.DBX 13.0;
      A     I 1.5;
      =     DB82.DBX 13.6;
      A     I 3.5;
      =     DB82.DBX 15.4;
      AN    M 135.0;
      A     M 135.1;
      JC    M001;
      A     I 4.1;
      AN    DB21.DBX 35.0;
      A     I 32.0;
      =     DB82.DBX 13.7;
      A     I 5.1;
      AN    DB21.DBX 35.0;
      A     I 32.0;
      =     DB82.DBX 14.0;
M001: NOP   0;
      A     I 5.2;
      A     I 32.0;
      =     DB82.DBX 16.0;
      A     I 1.2;
      =     DB82.DBX 14.5;
      A     I 1.1;
      =     DB82.DBX 14.4;
      A     I 1.0;
      =     DB82.DBX 14.3;
      A     I 6.4;
      =     DB82.DBX 14.6;
      A     I 6.5;
      =     DB82.DBX 14.7;
      A     DB82.DBX 42.5;
      AN    DB82.DBX 42.7;
      O;
      AN    DB82.DBX 42.5;
      A     DB82.DBX 42.7;
      S     M 83.0;
      A     I 6.3;
      AN    M 83.0;
      O;
      A     I 6.3;
      A     M 83.0;
      AN    DB82.DBX 42.5;
      A     DB82.DBX 42.7;
      O;
      A     M 135.1;
      A     I 5.1;
      A     Q 4.3;
      =     DB82.DBX 15.1;
      A     I 6.3;
      AN    M 83.0;
      O;
      A     I 6.3;
      A     M 83.0;
      A     DB82.DBX 42.5;
      AN    DB82.DBX 42.7;
      O;
      A     M 135.1;
      A     I 5.1;
      A     Q 4.3;
      =     DB82.DBX 15.3;
      A     I 6.3;
      A(;
      A     DB82.DBX 42.5;
      A     DB82.DBX 42.7;
      O;
      AN    DB82.DBX 42.5;
      AN    DB82.DBX 42.7;
      );
      R     M 83.0;
      A     I 6.6;
      A(;
      O     DB82.DBX 42.4;
      O     DB21.DBX 35.0;
      );
      =     DB82.DBX 15.0;
      L     1;
      T     DB82.DBB 17;
      A     I 6.2;
      =     DB82.DBX 15.5;
      A     I 6.1;
      =     DB82.DBX 15.6;
      A     I 3.7;
      =     DB82.DBX 16.3;
      A     DB82.DBX 40.1;
      =     Q 5.0;
      A     DB82.DBX 40.2;
      =     Q 5.6;
      A     DB82.DBX 40.5;
      =     Q 5.2;
      A     DB82.DBX 40.6;
      =     Q 5.4;
      A     DB82.DBX 41.1;
      =     Q 5.5;
      A     DB82.DBX 41.2;
      =     Q 5.1;
      A     DB82.DBX 41.3;
      A     DB82.DBX 41.7;
      AN    DB82.DBX 42.0;
      =     Q 3.5;
      A     DB82.DBX 41.4;
      A     DB82.DBX 41.7;
      AN    DB82.DBX 42.0;
      =     Q 2.3;
      A     DB82.DBX 42.0;
      =     Q 3.4;
      A     DB82.DBX 41.5;
      =     Q 1.5;
      A     DB82.DBX 41.6;
      =     Q 1.4;
      A     DB82.DBX 43.1;
      =     Q 2.2;
      A     DB82.DBX 42.3;
      =     Q 0.6;
      A     DB82.DBX 42.2;
      =     Q 0.5;
      A     DB82.DBX 42.1;
      =     Q 0.4;
      A     DB82.DBX 42.4;
      =     Q 4.6;
      A     DB82.DBX 42.5;
      A     DB82.DBX 42.7;
      =     Q 4.3;
      A     I 2.5;
      O;
      A(;
      O     I 7.1;
      O     M 40.0;
      );
      AN    Q 3.5;
      AN    Q 2.3;
      R     Q 2.0;
      S     Q 2.1;
      AN    I 2.4;
      S     Q 2.0;
      R     Q 2.1;
      A     Q 2.0;
      =     DB33.DBX 4.3;
      A     I 2.3;
      R     Q 1.6;
      S     Q 1.7;
      AN    I 2.2;
      S     Q 1.6;
      R     Q 1.7;
      A     Q 1.6;
      =     DB21.DBX 6.0;
      =     DB21.DBX 6.1;
END_FUNCTION

FUNCTION FC 91 : VOID
AUTHOR : Tested
NAME : Logic
VERSION : 0.2
BEGIN
// (block stored without names or comments; labels and parameter names are numbered)
NETWORK
TITLE =
      A     DB82.DBX 40.0;
      FP    M 90.3;
      =     M 90.4;
      AN    M 90.4;
      JC    M001;
      R     M 83.1;
      R     M 83.2;
      R     M 83.6;
      R     Q 3.2;
      R     DB21.DBX 20.0;
      R     DB21.DBX 20.1;
      R     DB21.DBX 20.2;
M001: AN    DB82.DBX 40.0;
      JC    M003;
NETWORK
TITLE =
      A     I 6.3;
      AN    M 83.7;
      =     M 90.0;
      A     I 6.3;
      =     M 83.7;
NETWORK
TITLE =
      A     M 135.0;
      ON    M 135.1;
      JC    M002;
      A     I 5.1;
      AN    M 83.4;
      =     M 83.5;
      A     I 5.1;
      =     M 83.4;
NETWORK
TITLE =
      O     M 83.5;
      O     M 90.0;
      A     Q 3.2;
      R     M 83.6;
      A     M 83.5;
      AN    Q 3.2;
      S     M 83.6;
      A     M 83.6;
      =     Q 3.2;
NETWORK
TITLE =
      A     DB82.DBX 40.0;
      A     Q 3.2;
      A     I 4.3;
      S     M 83.1;
      O     I 5.7;
      ON    Q 3.2;
      R     M 83.1;
NETWORK
TITLE =
      A     DB82.DBX 40.0;
      A     Q 3.2;
      A     I 5.7;
      S     M 83.2;
      O     I 4.3;
      ON    Q 3.2;
      R     M 83.2;
NETWORK
TITLE =
      A     DB82.DBX 40.0;
      A     M 83.1;
      =     Q 2.6;
      R     DB21.DBX 12.0;
      R     DB21.DBX 12.1;
      S     DB21.DBX 12.2;
NETWORK
TITLE =
      A     DB82.DBX 40.0;
      A     M 83.2;
      =     Q 4.0;
      R     DB21.DBX 20.0;
      R     DB21.DBX 20.1;
      S     DB21.DBX 20.2;
M002: NOP   0;
NETWORK
TITLE =
M003: A     DB82.DBX 40.0;
      FN    M 90.1;
      =     M 90.2;
      AN    M 90.2;
      JC    M004;
      R     M 83.1;
      R     M 83.2;
      R     M 83.6;
      R     Q 3.2;
      R     DB21.DBX 20.0;
      R     DB21.DBX 20.1;
      R     DB21.DBX 20.2;
M004: A     DB82.DBX 40.0;
      JC    M005;
NETWORK
TITLE =
      AN    DB82.DBX 40.0;
      A     DB10.DBX 100.7;
      A     DB10.DBX 100.6;
      A     DB10.DBX 100.0;
      AN    DB10.DBX 100.1;
      AN    DB10.DBX 100.2;
      AN    DB10.DBX 100.3;
      AN    DB10.DBX 100.4;
      =     DB31.DBX 4.0;
NETWORK
TITLE =
      AN    DB82.DBX 40.0;
      A     DB10.DBX 101.7;
      A     DB10.DBX 101.6;
      AN    DB10.DBX 101.0;
      A     DB10.DBX 101.1;
      AN    DB10.DBX 101.2;
      AN    DB10.DBX 101.3;
      AN    DB10.DBX 101.4;
      =     DB32.DBX 4.1;
NETWORK
TITLE =
      A     M 135.0;
      ON    M 135.1;
      JC    M005;
      A     DB10.DBX 102.7;
      A     DB10.DBX 102.6;
      A     DB10.DBX 102.0;
      AN    DB10.DBX 102.1;
      AN    DB10.DBX 102.2;
      AN    DB10.DBX 102.3;
      AN    DB10.DBX 102.4;
      =     DB31.DBX 4.2;
NETWORK
TITLE =
      A     DB10.DBX 102.7;
      A     DB10.DBX 102.6;
      AN    DB10.DBX 102.0;
      A     DB10.DBX 102.1;
      AN    DB10.DBX 102.2;
      AN    DB10.DBX 102.3;
      AN    DB10.DBX 102.4;
      =     DB32.DBX 4.2;
NETWORK
TITLE =
M005: NOP   0;
END_FUNCTION

DATA_BLOCK DB 1
VERSION : 0.1
BEGIN
// 6300 bytes; values not shown
END_DATA_BLOCK

DATA_BLOCK DB 2
VERSION : 0.0
BEGIN
// 196 bytes; values not shown
END_DATA_BLOCK

DATA_BLOCK DB 3
VERSION : 0.0
BEGIN
// 196 bytes; values not shown
END_DATA_BLOCK

DATA_BLOCK DB 4
AUTHOR : NUMERIK
FAMILY : _800D
NAME : Basics
VERSION : 2.0
BEGIN
// 226 bytes; values not shown
END_DATA_BLOCK

DATA_BLOCK DB 5
AUTHOR : NUMERIK
FAMILY : _800D
NAME : Basics
VERSION : 2.6
BEGIN
// 262 bytes; values not shown
END_DATA_BLOCK

DATA_BLOCK DB 6
VERSION : 0.0
BEGIN
// 272 bytes; values not shown
END_DATA_BLOCK

DATA_BLOCK DB 7
AUTHOR : NUMERIK
FAMILY : _800D
NAME : Basics
VERSION : 2.2
FB 1
BEGIN
END_DATA_BLOCK

DATA_BLOCK DB 8
AUTHOR : NUMERIK
FAMILY : _800D
NAME : Basics
VERSION : 4.1
BEGIN
// 166 bytes; values not shown
END_DATA_BLOCK

DATA_BLOCK DB 10
AUTHOR : NUMERIK
FAMILY : _800D
NAME : Basics
VERSION : 1.1
UDT 10
BEGIN
END_DATA_BLOCK

DATA_BLOCK DB 11
VERSION : 0.0
BEGIN
// 20 bytes; values not shown
END_DATA_BLOCK

DATA_BLOCK DB 15
AUTHOR : NUMERIK
FAMILY : _800D
NAME : Bas_Com
VERSION : 2.0
FB 6
BEGIN
END_DATA_BLOCK

// DB 16: know-how protected block, not included

DATA_BLOCK DB 17
AUTHOR : NUMERIK
FAMILY : _800D
NAME : Basics
VERSION : 2.0
BEGIN
// 4 bytes; values not shown
END_DATA_BLOCK

DATA_BLOCK DB 18
AUTHOR : NUMERIK
FAMILY : _800D
NAME : Basics
VERSION : 1.1
BEGIN
// 128 bytes; values not shown
END_DATA_BLOCK

DATA_BLOCK DB 19
AUTHOR : NUMERIK
FAMILY : _800D
NAME : Basics
VERSION : 2.1
UDT 19
BEGIN
END_DATA_BLOCK

DATA_BLOCK DB 20
VERSION : 0.0
BEGIN
// 40 bytes; values not shown
END_DATA_BLOCK

DATA_BLOCK DB 21
VERSION : 0.0
BEGIN
// 364 bytes; values not shown
END_DATA_BLOCK

DATA_BLOCK DB 31
VERSION : 0.0
BEGIN
// 112 bytes; values not shown
END_DATA_BLOCK

DATA_BLOCK DB 32
VERSION : 0.0
BEGIN
// 112 bytes; values not shown
END_DATA_BLOCK

DATA_BLOCK DB 33
VERSION : 0.0
BEGIN
// 112 bytes; values not shown
END_DATA_BLOCK

DATA_BLOCK DB 34
VERSION : 0.0
BEGIN
// 112 bytes; values not shown
END_DATA_BLOCK

DATA_BLOCK DB 70
AUTHOR : USER
VERSION : 5.2
BEGIN
// 10 bytes; values not shown
END_DATA_BLOCK

DATA_BLOCK DB 72
AUTHOR : USER
VERSION : 0.1
FB 120
BEGIN
END_DATA_BLOCK

// DB 81: know-how protected block, not included

DATA_BLOCK DB 82
AUTHOR : NUMERIK
NAME : SPSSS
VERSION : 5.3
BEGIN
// 198 bytes; values not shown
END_DATA_BLOCK

// DB 83: know-how protected block, not included

DATA_BLOCK DB 84
VERSION : 0.0
BEGIN
// 432 bytes; values not shown
END_DATA_BLOCK

DATA_BLOCK DB 85
VERSION : 0.0
BEGIN
// 426 bytes; values not shown
END_DATA_BLOCK

DATA_BLOCK DB 86
VERSION : 0.0
BEGIN
// 278 bytes; values not shown
END_DATA_BLOCK

DATA_BLOCK DB 87
VERSION : 0.0
BEGIN
// 450 bytes; values not shown
END_DATA_BLOCK

DATA_BLOCK DB 88
VERSION : 0.0
FB 28
BEGIN
END_DATA_BLOCK

DATA_BLOCK DB 90
AUTHOR : USER
VERSION : 0.1
FB 120
BEGIN
END_DATA_BLOCK

DATA_BLOCK DB 91
AUTHOR : USER
VERSION : 0.2
FB 3
BEGIN
END_DATA_BLOCK

DATA_BLOCK DB 100
VERSION : 0.1
BEGIN
// 2 bytes; values not shown
END_DATA_BLOCK

ORGANIZATION_BLOCK OB 1
VERSION : 2.0
BEGIN
// (block stored without names or comments; labels and parameter names are numbered)
NETWORK
TITLE =
      CALL  FC 2;
      L     LB 1;
      L     1;
      ==I;
      =     L 20.0;
      CALL  FC 30 (
           $1                       := L 20.0);
      A     L 20.0;
      S     I 0.7;
      S     I 1.5;
      A     DB82.DBX 40.0;
      FP    M 2.0;
      JCN   M001;
      L     0;
      T     QW 0;
      T     QW 2;
      T     QW 4;
      S     Q 1.4;
      S     Q 1.6;
      S     Q 2.0;
M001: A     DB82.DBX 40.0;
      FN    M 2.1;
      JCN   M002;
      L     0;
      T     QW 0;
      T     QW 2;
      T     QW 4;
      S     Q 1.4;
      S     Q 1.6;
      S     Q 2.0;
M002: AN    DB82.DBX 40.0;
      JC    M003;
      CALL  FC 90;
      JU    M004;
M003: CALL  FC 19 (
           $1                       := B#16#1,
           $2                       := B#16#1,
           $3                       := B#16#3,
           $4                       := P#M 22.0,
           $5                       := M 22.1);
      OPN   DB 21;
      O     M 22.0;
      =     DBX 6.0;
      OPN   DB 33;
      O     M 22.1;
      =     DBX 4.3;
      X     DB19.DBX 20.7;
      X     DB19.DBX 0.7;
      =     DB19.DBX 0.7;
      A     Q 1.6;
      =     DB21.DBX 6.1;
      SET;
M004: A     DB82.DBX 64.0;
      =     DB2.DBX 184.0;
      A     DB82.DBX 64.1;
      =     DB2.DBX 184.1;
      A     DB82.DBX 64.2;
      =     DB2.DBX 184.2;
      A     DB82.DBX 64.3;
      =     DB2.DBX 184.3;
      A     DB82.DBX 64.4;
      =     DB2.DBX 184.4;
      A     DB82.DBX 64.5;
      =     DB2.DBX 184.5;
      A     DB82.DBX 64.6;
      =     DB2.DBX 184.6;
      L     DB82.DBB 67;
      L     0;
      <>I;
      =     DB2.DBX 184.7;
      A     M 51.0;
      ON    M 51.0;
      =     M 51.0;
      CALL  FC 91;
      CALL  FC 52;
      A     M 134.0;
      JC    M005;
      CALL  FC 60;
M005: NOP   0;
      A     M 51.0;
      R     M 75.2;
      CALL  FC 10 (
           $1                       := FALSE,
           $2                       := I 3.7);
      BE;
END_ORGANIZATION_BLOCK

ORGANIZATION_BLOCK OB 35
AUTHOR : Zagorski
NAME : alarmpro
VERSION : 0.3
BEGIN
// (block stored without names or comments; labels and parameter names are numbered)
NETWORK
TITLE =
      A     M 126.0;
      JC    M026;
NETWORK
TITLE =
      L     PIB 32;
      T     IB 32;
NETWORK
TITLE =
      O     DB21.DBX 200.3;
      O     DB21.DBX 200.4;
      O     DB21.DBX 200.5;
      O     DB21.DBX 200.6;
      O     DB21.DBX 200.7;
      O     DB21.DBX 201.0;
      O     DB21.DBX 201.1;
      O     DB21.DBX 201.2;
      =     M 77.1;
NETWORK
TITLE =
      AN    DB21.DBX 200.3;
      AN    DB21.DBX 200.4;
      AN    DB21.DBX 200.5;
      AN    DB21.DBX 200.6;
      AN    DB21.DBX 200.7;
      AN    DB21.DBX 201.0;
      AN    DB21.DBX 201.1;
      AN    DB21.DBX 201.2;
      AN    DB21.DBX 201.3;
      AN    DB21.DBX 201.4;
      AN    DB21.DBX 201.5;
      AN    DB21.DBX 201.6;
      JC    M012;
      AN    DB21.DBX 200.3;
      JC    M001;
      L     256;
      T     MW 53;
      JU    M012;
M001: AN    DB21.DBX 200.4;
      JC    M002;
      L     512;
      T     MW 53;
      JU    M012;
M002: AN    DB21.DBX 200.5;
      JC    M003;
      L     1024;
      T     MW 53;
      JU    M012;
M003: AN    DB21.DBX 200.6;
      JC    M004;
      L     2048;
      T     MW 53;
      JU    M012;
M004: AN    DB21.DBX 200.7;
      JC    M005;
      L     4096;
      T     MW 53;
      JU    M012;
M005: AN    DB21.DBX 201.0;
      JC    M006;
      L     8192;
      T     MW 53;
      JU    M012;
M006: AN    DB21.DBX 201.1;
      JC    M007;
      L     16384;
      T     MW 53;
      JU    M012;
M007: AN    DB21.DBX 201.2;
      JC    M008;
      L     L#32768;
      T     MW 53;
      JU    M012;
M008: AN    DB21.DBX 201.3;
      JC    M009;
      L     1;
      T     MW 53;
      JU    M012;
M009: AN    DB21.DBX 201.4;
      JC    M010;
      L     2;
      T     MW 53;
      JU    M012;
M010: AN    DB21.DBX 201.5;
      JC    M011;
      L     4;
      T     MW 53;
      JU    M012;
M011: AN    DB21.DBX 201.6;
      JC    M012;
      L     8;
      T     MW 53;
M012: NOP   0;
NETWORK
TITLE =
      O     DB21.DBX 200.3;
      O     DB21.DBX 200.4;
      O     DB21.DBX 200.5;
      O     DB21.DBX 200.6;
      O     DB21.DBX 200.7;
      O     DB21.DBX 201.0;
      O     DB21.DBX 201.1;
      O     DB21.DBX 201.2;
      O     DB21.DBX 201.3;
      O     DB21.DBX 201.4;
      O     DB21.DBX 201.5;
      O     DB21.DBX 201.6;
      =     M 77.0;
NETWORK
TITLE =
      A     M 77.0;
      AN    DB21.DBX 200.3;
      AN    DB21.DBX 200.4;
      AN    DB21.DBX 200.5;
      AN    DB21.DBX 200.6;
      AN    DB21.DBX 200.7;
      AN    DB21.DBX 201.0;
      AN    DB21.DBX 201.1;
      AN    DB21.DBX 201.2;
      S     M 77.5;
      A(;
      ON    M 39.0;
      O     M 75.1;
      O     M 75.2;
      );
      R     M 77.5;
      NOP   0;
NETWORK
TITLE =
      L     IB 32;
      L     2#111100;
      AW;
      SRW   2;
      T     MB 80;
NETWORK
TITLE =
      AN    M 53.0;
      JC    M013;
      L     1;
      T     MW 86;
      JU    M021;
M013: AN    M 53.1;
      JC    M014;
      L     2;
      T     MW 86;
      JU    M021;
M014: AN    M 53.2;
      JC    M015;
      L     3;
      T     MW 86;
      JU    M021;
M015: AN    M 53.3;
      JC    M016;
      L     4;
      T     MW 86;
      JU    M021;
M016: AN    M 53.4;
      JC    M017;
      L     5;
      T     MW 86;
      JU    M021;
M017: AN    M 53.5;
      JC    M018;
      L     6;
      T     MW 86;
      JU    M021;
M018: AN    M 53.6;
      JC    M019;
      L     7;
      T     MW 86;
      JU    M021;
M019: AN    M 53.7;
      JC    M020;
      L     8;
      T     MW 86;
      JU    M021;
M020: L     0;
      T     MW 86;
      A     M 51.0;
      S     M 76.0;
M021: ON    M 39.0;
      O     M 75.1;
      R     M 76.0;
NETWORK
TITLE =
      L     MB 80;
      L     MB 87;
      ==I;
      A     I 32.6;
      =     M 77.4;
NETWORK
TITLE =
      L     MB 87;
      L     MB 80;
      -I;
      T     MW 92;
NETWORK
TITLE =
      L     MW 92;
      L     4;
      >I;
      =     M 89.0;
NETWORK
TITLE =
      L     MW 92;
      L     0;
      <=I;
      =     M 89.6;
NETWORK
TITLE =
      L     MW 92;
      L     -4;
      >=I;
      =     M 89.1;
NETWORK
TITLE =
      A     M 77.1;
      R     M 89.2;
      A     M 77.1;
      A(;
      O     M 89.0;
      O;
      A     M 89.1;
      A     M 89.6;
      );
      S     M 89.2;
      NOP   0;
NETWORK
TITLE =
NETWORK
TITLE =
      AN    M 89.2;
      JC    M022;
      L     MB 87;
      L     1;
      -I;
      T     MB 84;
      JU    M023;
M022: L     MB 87;
      L     1;
      +I;
      T     MB 84;
M023: L     MB 84;
      L     9;
      <I;
      JC    M024;
      L     1;
      T     MB 84;
M024: L     MB 84;
      L     0;
      <>I;
      JC    M025;
      L     8;
      T     MB 84;
M025: NOP   0;
NETWORK
TITLE =
      L     MB 84;
      L     MB 80;
      ==I;
      =     M 89.7;
NETWORK
TITLE =
      A(;
      O     Q 37.0;
      O     Q 37.1;
      O     Q 37.2;
      );
      L     S5T#4S;
      SD    T 81;
      NOP   0;
      NOP   0;
      NOP   0;
      NOP   0;
NETWORK
TITLE =
      A     T 81;
      S     M 76.3;
      A     I 3.7;
      R     M 76.3;
      NOP   0;
NETWORK
TITLE =
      A     M 77.4;
      S     M 89.5;
      A(;
      O     Q 37.2;
      O     M 77.1;
      );
      R     M 89.5;
      NOP   0;
NETWORK
TITLE =
      A     I 32.6;
      FN    M 69.0;
      =     M 69.1;
NETWORK
TITLE =
      A     I 32.6;
      FP    M 69.2;
      =     M 69.3;
NETWORK
TITLE =
      A     M 75.5;
      L     S5T#3S;
      SE    T 80;
      NOP   0;
      NOP   0;
      NOP   0;
      A     T 80;
      =     M 75.3;
NETWORK
TITLE =
      A     M 69.1;
      A(;
      O     M 89.5;
      O     M 75.3;
      );
      S     Q 37.2;
      A(;
      AN    M 75.5;
      A     M 69.3;
      A     Q 37.2;
      O     M 77.5;
      O     M 76.3;
      );
      R     Q 37.2;
      NOP   0;
NETWORK
TITLE =
      A(;
      A(;
      A     M 89.2;
      A(;
      A     M 77.1;
      AN    M 77.4;
      O     M 75.5;
      );
      O     Q 37.1;
      );
      A     I 33.2;
      O;
      A(;
      AN    M 89.2;
      AN    M 75.3;
      O;
      AN    M 88.2;
      A     M 75.3;
      );
      AN    I 33.2;
      A     Q 37.2;
      );
      AN    M 76.3;
      AN    M 77.5;
      AN    Q 37.0;
      A     I 32.0;
      =     Q 37.1;
NETWORK
TITLE =
      A(;
      A(;
      AN    M 89.2;
      A(;
      A     M 77.1;
      AN    M 77.4;
      O     M 75.5;
      );
      O     Q 37.0;
      );
      A     I 33.2;
      O;
      A(;
      A     M 89.2;
      AN    M 75.3;
      O;
      A     M 88.2;
      A     M 75.3;
      );
      AN    I 33.2;
      A     Q 37.2;
      );
      AN    M 76.3;
      AN    M 77.5;
      AN    Q 37.1;
      A     I 32.0;
      =     Q 37.0;
NETWORK
TITLE =
      A     Q 37.1;
      AN    M 75.3;
      S     M 88.2;
      A     Q 37.0;
      AN    M 75.3;
      R     M 88.2;
      NOP   0;
NETWORK
TITLE =
      A     I 33.2;
      AN    Q 37.2;
      AN    Q 37.1;
      AN    Q 37.0;
      =     M 88.4;
NETWORK
TITLE =
      A     M 75.5;
      S     M 75.4;
      A     M 77.1;
      R     M 75.4;
      NOP   0;
NETWORK
TITLE =
      A(;
      A(;
      A     I 32.2;
      AN    I 32.3;
      O;
      AN    I 32.2;
      A     I 32.3;
      );
      AN    I 32.4;
      AN    I 32.5;
      O;
      A(;
      AN    I 32.2;
      AN    I 32.3;
      O;
      A     I 32.2;
      A     I 32.3;
      );
      A(;
      A     I 32.4;
      AN    I 32.5;
      O;
      AN    I 32.4;
      A     I 32.5;
      );
      );
      A     I 32.6;
      =     M 88.1;
NETWORK
TITLE =
      A(;
      A     M 88.1;
      AN    I 32.7;
      O;
      AN    M 88.1;
      A     I 32.7;
      );
      S     M 76.7;
      A(;
      ON    M 88.4;
      O     M 75.1;
      );
      R     M 76.7;
      NOP   0;
NETWORK
TITLE =
      ON    M 88.4;
      ON    M 77.4;
      O     M 76.7;
      =     M 76.2;
NETWORK
TITLE =
      A     M 76.2;
      AN    M 75.3;
      A(;
      A     DB82.DBX 40.0;
      AN    M 38.0;
      O;
      AN    DB82.DBX 40.0;
      AN    DB11.DBX 6.2;
      AN    DB11.DBX 7.2;
      );
      S     DB21.DBX 6.1;
NETWORK
TITLE =
      A     M 51.0;
      A     M 76.2;
      AN    M 75.3;
      A(;
      A     DB82.DBX 40.0;
      AN    M 38.0;
      O;
      AN    DB82.DBX 40.0;
      AN    DB11.DBX 6.2;
      AN    DB11.DBX 7.2;
      );
      S     DB21.DBX 6.0;
NETWORK
TITLE =
NETWORK
TITLE =
      L     QB 37;
      T     PQB 37;
NETWORK
TITLE =
NETWORK
TITLE =
      A     M 51.0;
      R     M 75.5;
NETWORK
TITLE =
M026: NOP   0;
END_ORGANIZATION_BLOCK

ORGANIZATION_BLOCK OB 40
VERSION : 4.11
BEGIN
// (block stored without names or comments; labels and parameter names are numbered)
NETWORK
TITLE =
      CALL  FC 3;
END_ORGANIZATION_BLOCK

ORGANIZATION_BLOCK OB 100
VERSION : 4.11
BEGIN
// (block stored without names or comments; labels and parameter names are numbered)
NETWORK
TITLE =
      CALL  FB 1 , DB 7 (
           DIW 0                    := 1,
           DIW 2                    := 0,
           DID 4                    := P#I 0.0,
           DIW 8                    := 0,
           DID 10                   := P#Q 0.0,
           DIW 14                   := 0,
           DID 16                   := P#Q 8.0,
           DIW 20                   := 0,
           DID 22                   := P#Q 12.0,
           DIW 26                   := 14,
           DIW 28                   := 112,
           DIW 30                   := 32,
           DIX 62.0                 := TRUE,
           DIW 110                  := 32,
           DIW 112                  := 5376,
           DIX 116.0                := TRUE,
           DIX 116.1                := TRUE,
           DIX 116.2                := FALSE,
           DIW 118                  := 2);
NETWORK
TITLE =
      L     DB20.DBW 4;
      L     0;
      ==I;
      =     M 125.0;
      L     DB20.DBW 4;
      L     1;
      ==I;
      =     M 125.1;
      L     DB20.DBW 4;
      L     2;
      ==I;
      =     M 125.2;
NETWORK
TITLE =
      L     DB20.DBW 6;
      L     0;
      ==I;
      =     M 126.0;
      L     DB20.DBW 6;
      L     1;
      ==I;
      =     M 126.1;
      L     DB20.DBW 6;
      L     2;
      ==I;
      =     M 126.2;
NETWORK
TITLE =
      L     DB20.DBW 12;
      L     0;
      ==I;
      =     M 129.0;
      L     DB20.DBW 12;
      L     1;
      ==I;
      =     M 129.1;
      L     DB20.DBW 12;
      L     2;
      ==I;
      =     M 129.2;
NETWORK
TITLE =
      L     DB20.DBW 22;
      L     0;
      ==I;
      =     M 134.0;
      L     DB20.DBW 22;
      L     1;
      ==I;
      =     M 134.1;
      L     DB20.DBW 22;
      L     2;
      ==I;
      =     M 134.2;
      L     DB20.DBW 22;
      L     3;
      ==I;
      =     M 134.3;
      L     DB20.DBW 22;
      L     4;
      ==I;
      =     M 134.4;
NETWORK
TITLE =
      O     M 75.2;
      ON    M 75.2;
      S     M 75.2;
      O     M 75.5;
      ON    M 75.5;
      S     M 75.5;
END_ORGANIZATION_BLOCK
